Fanuc KAREL source: V_SNAP_VIEW.kl

PROGRAM T
%NOLOCKGROUP
VAR
 v0 : STRING[40]
 v1 : INTEGER
 v2 : INTEGER
 v3 : INTEGER
BEGIN
 V_SNAP_VIEW(v0, v1, v2, v3)
END T
